// LS Electric XG5000 project: 유튜브방송용_2021082621
// PLC NewPLC

PROGRAM NewProgram (task: 스캔 프로그램)

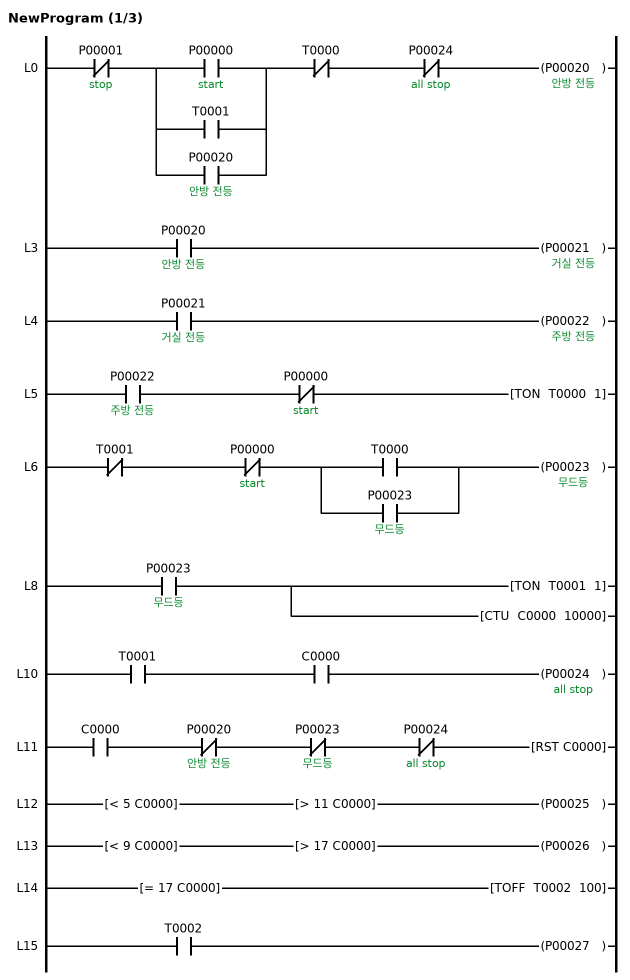
; L0
LOAD NOT  P00001	// stop
LOAD      P00000	// start
OR        T0001
OR        P00020	// 안방 전등
AND LOAD
AND NOT   T0000
AND NOT   P00024	// all stop
OUT       P00020	// 안방 전등
; L3
LOAD      P00020	// 안방 전등
OUT       P00021	// 거실 전등
; L4
LOAD      P00021	// 거실 전등
OUT       P00022	// 주방 전등
; L5
LOAD      P00022	// 주방 전등
AND NOT   P00000	// start
TON       T0000 1
; L6
LOAD NOT  T0001
AND NOT   P00000	// start
LOAD      T0000
OR        P00023	// 무드등
AND LOAD
OUT       P00023	// 무드등
; L8
LOAD      P00023	// 무드등
TON       T0001 1
CTU       C0000 10000
; L10
LOAD      T0001
AND       C0000
OUT       P00024	// all stop
; L11
LOAD      C0000
AND NOT   P00020	// 안방 전등
AND NOT   P00023	// 무드등
AND NOT   P00024	// all stop
RST       C0000
; L12
LOAD<     5 C0000
AND>      11 C0000
OUT       P00025
; L13
LOAD<     9 C0000
AND>      17 C0000
OUT       P00026
; L14
LOAD=     17 C0000
TOFF      T0002 100
; L15
LOAD      T0002
OUT       P00027

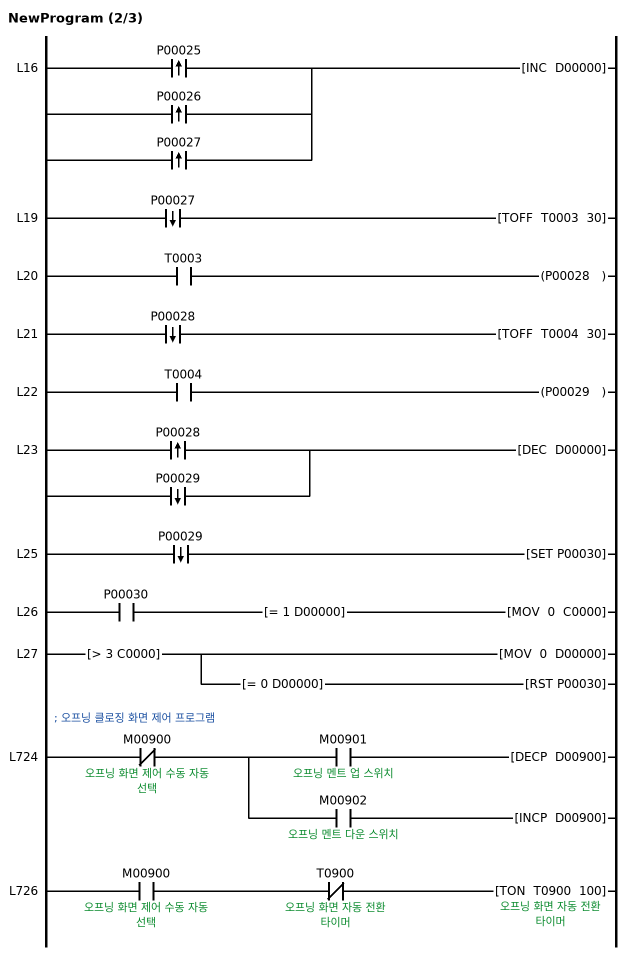
; L16
LOADP     P00025
ORP       P00026
ORP       P00027
INC       D00000
; L19
LOADN     P00027
TOFF      T0003 30
; L20
LOAD      T0003
OUT       P00028
; L21
LOADN     P00028
TOFF      T0004 30
; L22
LOAD      T0004
OUT       P00029
; L23
LOADP     P00028
ORN       P00029
DEC       D00000
; L25
LOADN     P00029
SET       P00030
; L26
LOAD      P00030
AND=      1 D00000
MOV       0 C0000
; L27
LOAD>     3 C0000
MOV       0 D00000
AND=      0 D00000
RST       P00030
// 오프닝 클로징 화면 제어 프로그램
; L724
LOAD NOT  M00900	// 오프닝 화면 제어 수동 자동 선택
MPUSH
AND       M00901	// 오프닝 멘트 업 스위치
DECP      D00900
MPOP
AND       M00902	// 오프닝 멘트 다운 스위치
INCP      D00900
; L726
LOAD      M00900	// 오프닝 화면 제어 수동 자동 선택
AND NOT   T0900	// 오프닝 화면 자동 전환 타이머
TON       T0900 100	// 오프닝 화면 자동 전환 타이머

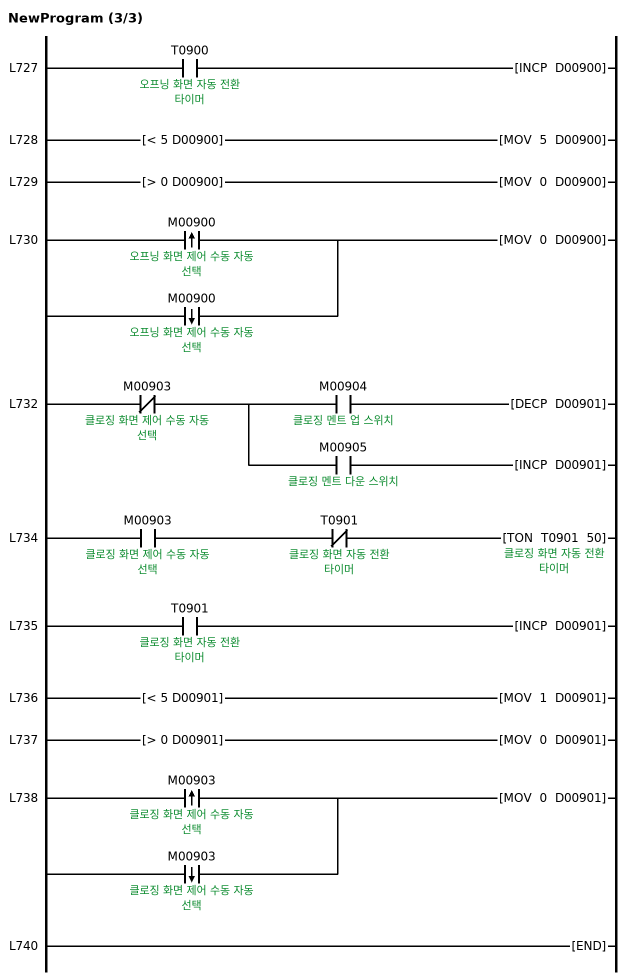
; L727
LOAD      T0900	// 오프닝 화면 자동 전환 타이머
INCP      D00900
; L728
LOAD<     5 D00900
MOV       5 D00900
; L729
LOAD>     0 D00900
MOV       0 D00900
; L730
LOADP     M00900	// 오프닝 화면 제어 수동 자동 선택
ORN       M00900	// 오프닝 화면 제어 수동 자동 선택
MOV       0 D00900
; L732
LOAD NOT  M00903	// 클로징 화면 제어 수동 자동 선택
MPUSH
AND       M00904	// 클로징 멘트 업 스위치
DECP      D00901
MPOP
AND       M00905	// 클로징 멘트 다운 스위치
INCP      D00901
; L734
LOAD      M00903	// 클로징 화면 제어 수동 자동 선택
AND NOT   T0901	// 클로징 화면 자동 전환 타이머
TON       T0901 50	// 클로징 화면 자동 전환 타이머
; L735
LOAD      T0901	// 클로징 화면 자동 전환 타이머
INCP      D00901
; L736
LOAD<     5 D00901
MOV       1 D00901
; L737
LOAD>     0 D00901
MOV       0 D00901
; L738
LOADP     M00903	// 클로징 화면 제어 수동 자동 선택
ORN       M00903	// 클로징 화면 제어 수동 자동 선택
MOV       0 D00901
; L740
END

VARIABLES AND COMMENTS (devices not used above)
P00002	BIT	주방 스위치